FUNCTION_BLOCK STATE_CHECK
  {SET_ATTRIBUTE(OpcUa, SERVICE)}
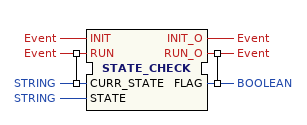
  EVENT_INPUT
    INIT;
    RUN WITH CURR_STATE;
  END_EVENT
  EVENT_OUTPUT
    INIT_O;
    RUN_O WITH FLAG;
  END_EVENT
  VAR_INPUT
    CURR_STATE : STRING;
    STATE : STRING;
  END_VAR
  VAR_OUTPUT
    FLAG : BOOLEAN;
  END_VAR
END_FUNCTION_BLOCK
